// TIA Portal V18 export
FUNCTION "DL_General" : Void   // FC51001, LAD
{ S7_Optimized_Access := 'TRUE' }
VERSION : 0.1
// stored: AutoNumber false, IsIECCheckEnabled false, SetENOAutomatically false, UDAEnableTagReadback false
   VAR_TEMP
      LvlRequest : Array[1..2] of Bool;
      xStopTriger : Bool;
      xCounter1Triger : Bool;
      xCounter2Triger : Bool;
      xPump1ExeriseRun : Bool;
      xPump2ExeriseRun : Bool;
      xPump1ExeriseRunTriger : Bool;
      xPump2ExeriseRunTriger : Bool;
      tTimeExericePump1 : Time;
      tTimeExericePump2 : Time;
   END_VAR
   VAR_TEMP   // added for the SCL form of the ladder/FBD networks
      _w1 : Bool;
      _w2 : Bool;
      _w3 : Bool;
      _w4 : Bool;
      _w5 : Bool;
      _w6 : Bool;
   END_VAR
BEGIN

REGION Network 1 (SCL): PanelModeSelector
   IF "DLsDI".Requests.xDieselLinePumpPanelSelectorAuto THEN
       "DL_Vars".Vars.cDLPanelModeSelector := 3;
   ELSIF "DLsDI".Requests.xDieselLinePumpPanelSelectorP1Man THEN
       "DL_Vars".Vars.cDLPanelModeSelector := 1;
   ELSIF "DLsDI".Requests.xDieselLinePumpPanelSelectorP2Man THEN
       "DL_Vars".Vars.cDLPanelModeSelector := 2;
   ELSIF "DLsDI".Requests.xDieselLinePumpPanelSelectorOff THEN
       "DL_Vars".Vars.cDLPanelModeSelector := 0;
   END_IF;
END_REGION

REGION Network 2
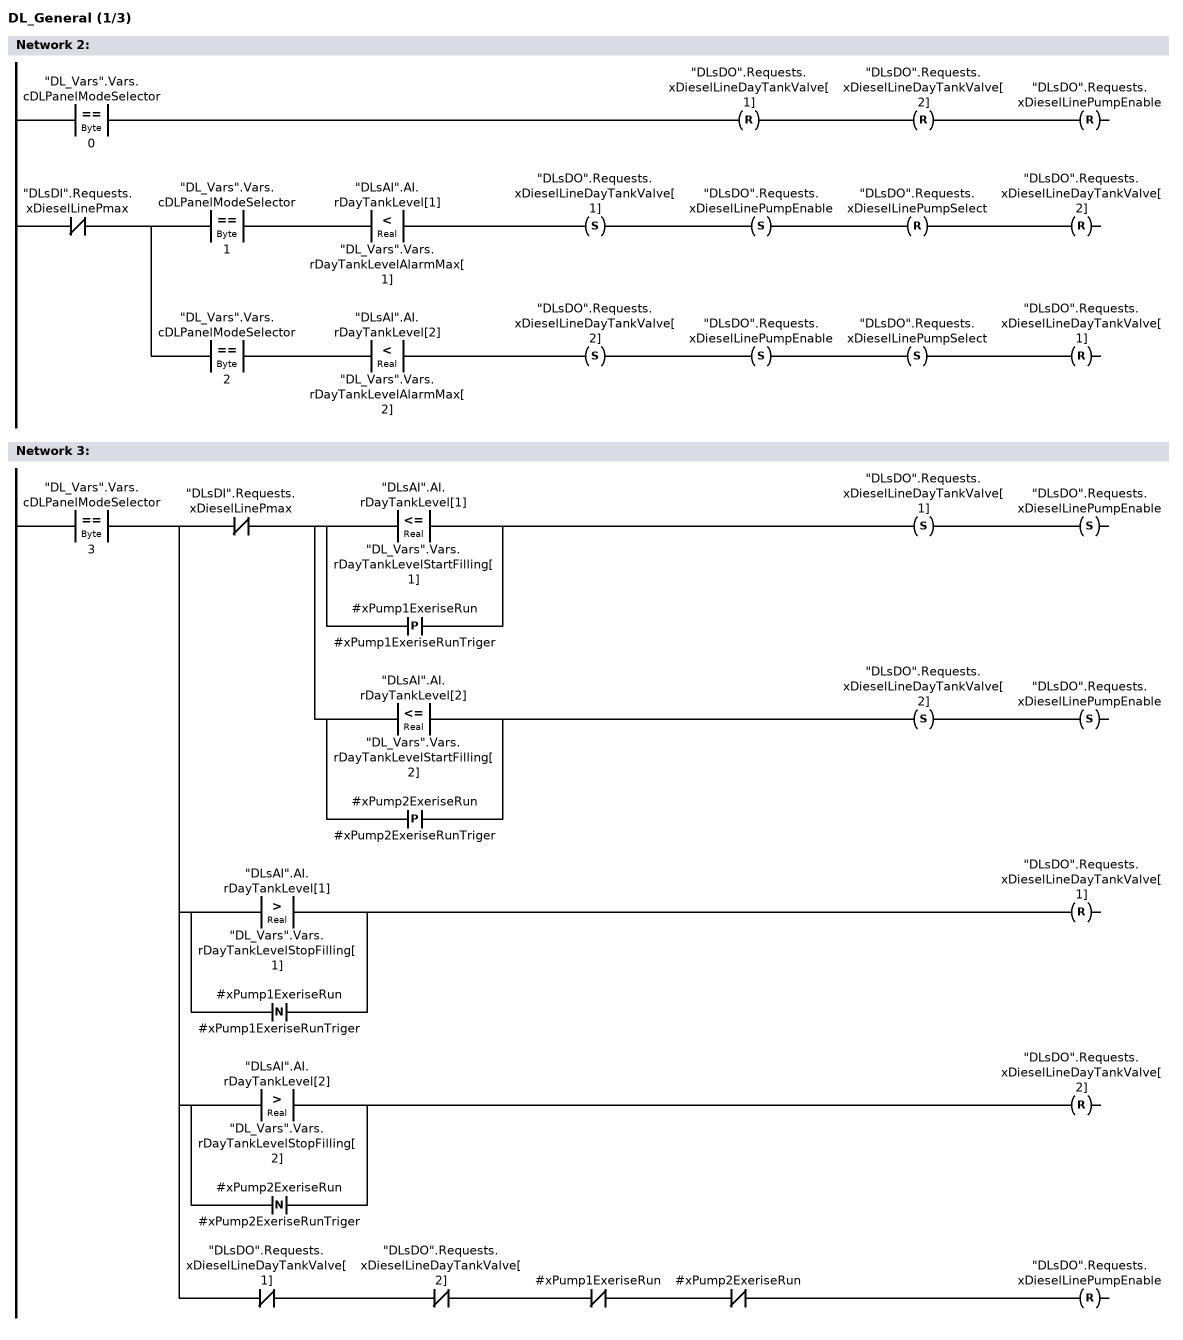
   RUNG wire#powerrail
      { S7_Templates := "SrcType := Byte" } EQ_Contact(in1 := "DL_Vars".Vars.cDLPanelModeSelector, in2 := 0)
      R_Coil( "DLsDO".Requests.xDieselLineDayTankValve[1] )
      R_Coil( "DLsDO".Requests.xDieselLineDayTankValve[2] )
      R_Coil( "DLsDO".Requests.xDieselLinePumpEnable )
   END_RUNG
   RUNG wire#powerrail
      I_Contact( "DLsDI".Requests.xDieselLinePmax )
      wire#w1
      { S7_Templates := "SrcType := Byte" } EQ_Contact(in1 := "DL_Vars".Vars.cDLPanelModeSelector, in2 := 1)
      { S7_Templates := "SrcType := Real" } LT_Contact(in1 := "DLsAI".AI.rDayTankLevel[1], in2 := "DL_Vars".Vars.rDayTankLevelAlarmMax[1])
      S_Coil( "DLsDO".Requests.xDieselLineDayTankValve[1] )
      S_Coil( "DLsDO".Requests.xDieselLinePumpEnable )
      R_Coil( "DLsDO".Requests.xDieselLinePumpSelect )
      R_Coil( "DLsDO".Requests.xDieselLineDayTankValve[2] )
   END_RUNG
   RUNG wire#w1
      { S7_Templates := "SrcType := Byte" } EQ_Contact(in1 := "DL_Vars".Vars.cDLPanelModeSelector, in2 := 2)
      { S7_Templates := "SrcType := Real" } LT_Contact(in1 := "DLsAI".AI.rDayTankLevel[2], in2 := "DL_Vars".Vars.rDayTankLevelAlarmMax[2])
      S_Coil( "DLsDO".Requests.xDieselLineDayTankValve[2] )
      S_Coil( "DLsDO".Requests.xDieselLinePumpEnable )
      S_Coil( "DLsDO".Requests.xDieselLinePumpSelect )
      R_Coil( "DLsDO".Requests.xDieselLineDayTankValve[1] )
   END_RUNG
   // the same network as SCL:
   IF "DL_Vars".Vars.cDLPanelModeSelector = 0 THEN
       "DLsDO".Requests.xDieselLineDayTankValve[1] := FALSE;
       "DLsDO".Requests.xDieselLineDayTankValve[2] := FALSE;
       "DLsDO".Requests.xDieselLinePumpEnable := FALSE;
   END_IF;
   #_w1 := NOT "DLsDI".Requests.xDieselLinePmax;
   IF #_w1 AND ("DL_Vars".Vars.cDLPanelModeSelector = 1) AND ("DLsAI".AI.rDayTankLevel[1] < "DL_Vars".Vars.rDayTankLevelAlarmMax[1]) THEN
       "DLsDO".Requests.xDieselLineDayTankValve[1] := TRUE;
       "DLsDO".Requests.xDieselLinePumpEnable := TRUE;
       "DLsDO".Requests.xDieselLinePumpSelect := FALSE;
       "DLsDO".Requests.xDieselLineDayTankValve[2] := FALSE;
   END_IF;
   IF #_w1 AND ("DL_Vars".Vars.cDLPanelModeSelector = 2) AND ("DLsAI".AI.rDayTankLevel[2] < "DL_Vars".Vars.rDayTankLevelAlarmMax[2]) THEN
       "DLsDO".Requests.xDieselLineDayTankValve[2] := TRUE;
       "DLsDO".Requests.xDieselLinePumpEnable := TRUE;
       "DLsDO".Requests.xDieselLinePumpSelect := TRUE;
       "DLsDO".Requests.xDieselLineDayTankValve[1] := FALSE;
   END_IF;
END_REGION

REGION Network 3
   RUNG wire#powerrail
      { S7_Templates := "SrcType := Byte" } EQ_Contact(in1 := "DL_Vars".Vars.cDLPanelModeSelector, in2 := 3)
      wire#w1
      I_Contact( "DLsDI".Requests.xDieselLinePmax )
      wire#w2
      { S7_Templates := "SrcType := Real" } LE_Contact(in1 := "DLsAI".AI.rDayTankLevel[1], in2 := "DL_Vars".Vars.rDayTankLevelStartFilling[1])
      wire#w3
      S_Coil( "DLsDO".Requests.xDieselLineDayTankValve[1] )
      S_Coil( "DLsDO".Requests.xDieselLinePumpEnable )
   END_RUNG
   RUNG wire#w2
      P_Contact(operand := #xPump1ExeriseRun, bit := #xPump1ExeriseRunTriger)
   END_RUNG wire#w3
   RUNG wire#w2
      { S7_Templates := "SrcType := Real" } LE_Contact(in1 := "DLsAI".AI.rDayTankLevel[2], in2 := "DL_Vars".Vars.rDayTankLevelStartFilling[2])
      wire#w4
      S_Coil( "DLsDO".Requests.xDieselLineDayTankValve[2] )
      S_Coil( "DLsDO".Requests.xDieselLinePumpEnable )
   END_RUNG
   RUNG wire#w2
      P_Contact(operand := #xPump2ExeriseRun, bit := #xPump2ExeriseRunTriger)
   END_RUNG wire#w4
   RUNG wire#w1
      { S7_Templates := "SrcType := Real" } GT_Contact(in1 := "DLsAI".AI.rDayTankLevel[1], in2 := "DL_Vars".Vars.rDayTankLevelStopFilling[1])
      wire#w5
      R_Coil( "DLsDO".Requests.xDieselLineDayTankValve[1] )
   END_RUNG
   RUNG wire#w1
      N_Contact(operand := #xPump1ExeriseRun, bit := #xPump1ExeriseRunTriger)
   END_RUNG wire#w5
   RUNG wire#w1
      { S7_Templates := "SrcType := Real" } GT_Contact(in1 := "DLsAI".AI.rDayTankLevel[2], in2 := "DL_Vars".Vars.rDayTankLevelStopFilling[2])
      wire#w6
      R_Coil( "DLsDO".Requests.xDieselLineDayTankValve[2] )
   END_RUNG
   RUNG wire#w1
      N_Contact(operand := #xPump2ExeriseRun, bit := #xPump2ExeriseRunTriger)
   END_RUNG wire#w6
   RUNG wire#w1
      I_Contact( "DLsDO".Requests.xDieselLineDayTankValve[1] )
      I_Contact( "DLsDO".Requests.xDieselLineDayTankValve[2] )
      I_Contact( #xPump1ExeriseRun )
      I_Contact( #xPump2ExeriseRun )
      R_Coil( "DLsDO".Requests.xDieselLinePumpEnable )
   END_RUNG
   // the same network as SCL:
   #_w1 := "DL_Vars".Vars.cDLPanelModeSelector = 3;
   #_w2 := #_w1 AND NOT "DLsDI".Requests.xDieselLinePmax;
   #_w3 := #_w2 AND #xPump1ExeriseRun AND NOT #xPump1ExeriseRunTriger;   // rising edge of #xPump1ExeriseRun
   #xPump1ExeriseRunTriger := #xPump1ExeriseRun;
   IF (#_w2 AND ("DLsAI".AI.rDayTankLevel[1] <= "DL_Vars".Vars.rDayTankLevelStartFilling[1])) OR #_w3 THEN
       "DLsDO".Requests.xDieselLineDayTankValve[1] := TRUE;
       "DLsDO".Requests.xDieselLinePumpEnable := TRUE;
   END_IF;
   #_w4 := #_w2 AND #xPump2ExeriseRun AND NOT #xPump2ExeriseRunTriger;   // rising edge of #xPump2ExeriseRun
   #xPump2ExeriseRunTriger := #xPump2ExeriseRun;
   IF (#_w2 AND ("DLsAI".AI.rDayTankLevel[2] <= "DL_Vars".Vars.rDayTankLevelStartFilling[2])) OR #_w4 THEN
       "DLsDO".Requests.xDieselLineDayTankValve[2] := TRUE;
       "DLsDO".Requests.xDieselLinePumpEnable := TRUE;
   END_IF;
   #_w5 := #_w1 AND NOT #xPump1ExeriseRun AND #xPump1ExeriseRunTriger;   // falling edge of #xPump1ExeriseRun
   #xPump1ExeriseRunTriger := #xPump1ExeriseRun;
   IF (#_w1 AND ("DLsAI".AI.rDayTankLevel[1] > "DL_Vars".Vars.rDayTankLevelStopFilling[1])) OR #_w5 THEN
       "DLsDO".Requests.xDieselLineDayTankValve[1] := FALSE;
   END_IF;
   #_w6 := #_w1 AND NOT #xPump2ExeriseRun AND #xPump2ExeriseRunTriger;   // falling edge of #xPump2ExeriseRun
   #xPump2ExeriseRunTriger := #xPump2ExeriseRun;
   IF (#_w1 AND ("DLsAI".AI.rDayTankLevel[2] > "DL_Vars".Vars.rDayTankLevelStopFilling[2])) OR #_w6 THEN
       "DLsDO".Requests.xDieselLineDayTankValve[2] := FALSE;
   END_IF;
   IF #_w1 AND NOT "DLsDO".Requests.xDieselLineDayTankValve[1] AND NOT "DLsDO".Requests.xDieselLineDayTankValve[2] AND NOT #xPump1ExeriseRun AND NOT #xPump2ExeriseRun THEN
       "DLsDO".Requests.xDieselLinePumpEnable := FALSE;
   END_IF;
END_REGION

REGION Network 4
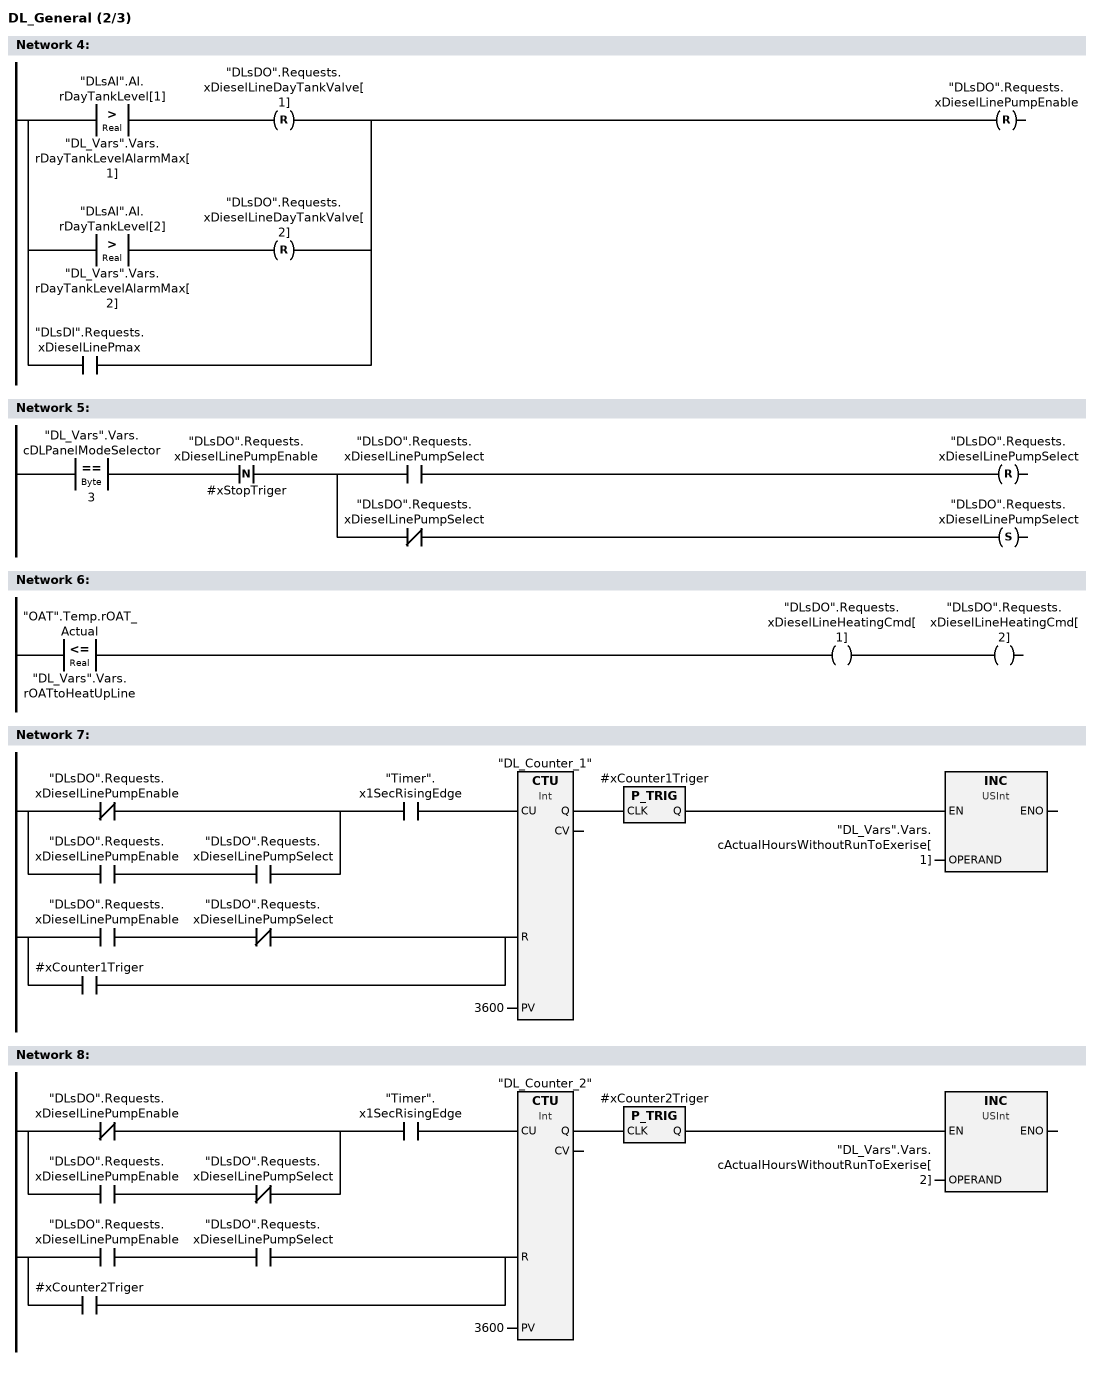
   RUNG wire#powerrail
      { S7_Templates := "SrcType := Real" } GT_Contact(in1 := "DLsAI".AI.rDayTankLevel[1], in2 := "DL_Vars".Vars.rDayTankLevelAlarmMax[1])
      R_Coil( "DLsDO".Requests.xDieselLineDayTankValve[1] )
      wire#w1
      R_Coil( "DLsDO".Requests.xDieselLinePumpEnable )
   END_RUNG
   RUNG wire#powerrail
      { S7_Templates := "SrcType := Real" } GT_Contact(in1 := "DLsAI".AI.rDayTankLevel[2], in2 := "DL_Vars".Vars.rDayTankLevelAlarmMax[2])
      R_Coil( "DLsDO".Requests.xDieselLineDayTankValve[2] )
   END_RUNG wire#w1
   RUNG wire#powerrail
      Contact( "DLsDI".Requests.xDieselLinePmax )
   END_RUNG wire#w1
   // the same network as SCL:
   #_w1 := "DLsAI".AI.rDayTankLevel[1] > "DL_Vars".Vars.rDayTankLevelAlarmMax[1];
   IF #_w1 THEN "DLsDO".Requests.xDieselLineDayTankValve[1] := FALSE; END_IF;
   #_w2 := "DLsAI".AI.rDayTankLevel[2] > "DL_Vars".Vars.rDayTankLevelAlarmMax[2];
   IF #_w2 THEN "DLsDO".Requests.xDieselLineDayTankValve[2] := FALSE; END_IF;
   IF #_w1 OR #_w2 OR "DLsDI".Requests.xDieselLinePmax THEN
       "DLsDO".Requests.xDieselLinePumpEnable := FALSE;
   END_IF;
END_REGION

REGION Network 5
   RUNG wire#powerrail
      { S7_Templates := "SrcType := Byte" } EQ_Contact(in1 := "DL_Vars".Vars.cDLPanelModeSelector, in2 := 3)
      N_Contact(operand := "DLsDO".Requests.xDieselLinePumpEnable, bit := #xStopTriger)
      wire#w1
      Contact( "DLsDO".Requests.xDieselLinePumpSelect )
      R_Coil( "DLsDO".Requests.xDieselLinePumpSelect )
   END_RUNG
   RUNG wire#w1
      I_Contact( "DLsDO".Requests.xDieselLinePumpSelect )
      S_Coil( "DLsDO".Requests.xDieselLinePumpSelect )
   END_RUNG
   // the same network as SCL:
   #_w1 := ("DL_Vars".Vars.cDLPanelModeSelector = 3) AND NOT "DLsDO".Requests.xDieselLinePumpEnable AND #xStopTriger;   // falling edge of "DLsDO".Requests.xDieselLinePumpEnable
   #xStopTriger := "DLsDO".Requests.xDieselLinePumpEnable;
   IF #_w1 AND "DLsDO".Requests.xDieselLinePumpSelect THEN
       "DLsDO".Requests.xDieselLinePumpSelect := FALSE;
   END_IF;
   IF #_w1 AND NOT "DLsDO".Requests.xDieselLinePumpSelect THEN
       "DLsDO".Requests.xDieselLinePumpSelect := TRUE;
   END_IF;
END_REGION

REGION Network 6
   RUNG wire#powerrail
      { S7_Templates := "SrcType := Real" } LE_Contact(in1 := "OAT".Temp.rOAT_Actual, in2 := "DL_Vars".Vars.rOATtoHeatUpLine)
      Coil( "DLsDO".Requests.xDieselLineHeatingCmd[1] )
      Coil( "DLsDO".Requests.xDieselLineHeatingCmd[2] )
   END_RUNG
   // the same network as SCL:
   "DLsDO".Requests.xDieselLineHeatingCmd[1] := "OAT".Temp.rOAT_Actual <= "DL_Vars".Vars.rOATtoHeatUpLine;
   "DLsDO".Requests.xDieselLineHeatingCmd[2] := "OAT".Temp.rOAT_Actual <= "DL_Vars".Vars.rOATtoHeatUpLine;
END_REGION

REGION Network 7
   RUNG wire#powerrail
      I_Contact( "DLsDO".Requests.xDieselLinePumpEnable )
      wire#w1
      Contact( "Timer".x1SecRisingEdge )
      { S7_Templates := "value_type := Int" } "DL_Counter_1".CTU(r := wire#w2, pv := 3600, cv =>)
      P_Trig( #xCounter1Triger )
      { S7_Templates := "DestType := USInt" } Inc( "DL_Vars".Vars.cActualHoursWithoutRunToExerise[1] )
   END_RUNG
   RUNG wire#powerrail
      Contact( "DLsDO".Requests.xDieselLinePumpEnable )
      Contact( "DLsDO".Requests.xDieselLinePumpSelect )
   END_RUNG wire#w1
   RUNG wire#powerrail
      Contact( "DLsDO".Requests.xDieselLinePumpEnable )
      I_Contact( "DLsDO".Requests.xDieselLinePumpSelect )
   END_RUNG wire#w2
   RUNG wire#powerrail
      Contact( #xCounter1Triger )
   END_RUNG wire#w2
   // the same network as SCL:
   "DL_Counter_1".CTU(CU := (NOT "DLsDO".Requests.xDieselLinePumpEnable OR ("DLsDO".Requests.xDieselLinePumpEnable AND "DLsDO".Requests.xDieselLinePumpSelect)) AND "Timer".x1SecRisingEdge,
                      R := ("DLsDO".Requests.xDieselLinePumpEnable AND NOT "DLsDO".Requests.xDieselLinePumpSelect) OR #xCounter1Triger,
                      PV := 3600);
   #_w1 := "DL_Counter_1".Q AND NOT #xCounter1Triger;   // rising edge
   #xCounter1Triger := "DL_Counter_1".Q;
   IF #_w1 THEN
       "DL_Vars".Vars.cActualHoursWithoutRunToExerise[1] := "DL_Vars".Vars.cActualHoursWithoutRunToExerise[1] + 1;
   END_IF;
END_REGION

REGION Network 8
   RUNG wire#powerrail
      I_Contact( "DLsDO".Requests.xDieselLinePumpEnable )
      wire#w1
      Contact( "Timer".x1SecRisingEdge )
      { S7_Templates := "value_type := Int" } "DL_Counter_2".CTU(r := wire#w2, pv := 3600, cv =>)
      P_Trig( #xCounter2Triger )
      { S7_Templates := "DestType := USInt" } Inc( "DL_Vars".Vars.cActualHoursWithoutRunToExerise[2] )
   END_RUNG
   RUNG wire#powerrail
      Contact( "DLsDO".Requests.xDieselLinePumpEnable )
      I_Contact( "DLsDO".Requests.xDieselLinePumpSelect )
   END_RUNG wire#w1
   RUNG wire#powerrail
      Contact( "DLsDO".Requests.xDieselLinePumpEnable )
      Contact( "DLsDO".Requests.xDieselLinePumpSelect )
   END_RUNG wire#w2
   RUNG wire#powerrail
      Contact( #xCounter2Triger )
   END_RUNG wire#w2
   // the same network as SCL:
   "DL_Counter_2".CTU(CU := (NOT "DLsDO".Requests.xDieselLinePumpEnable OR ("DLsDO".Requests.xDieselLinePumpEnable AND NOT "DLsDO".Requests.xDieselLinePumpSelect)) AND "Timer".x1SecRisingEdge,
                      R := ("DLsDO".Requests.xDieselLinePumpEnable AND "DLsDO".Requests.xDieselLinePumpSelect) OR #xCounter2Triger,
                      PV := 3600);
   #_w1 := "DL_Counter_2".Q AND NOT #xCounter2Triger;   // rising edge
   #xCounter2Triger := "DL_Counter_2".Q;
   IF #_w1 THEN
       "DL_Vars".Vars.cActualHoursWithoutRunToExerise[2] := "DL_Vars".Vars.cActualHoursWithoutRunToExerise[2] + 1;
   END_IF;
END_REGION

REGION Network 9
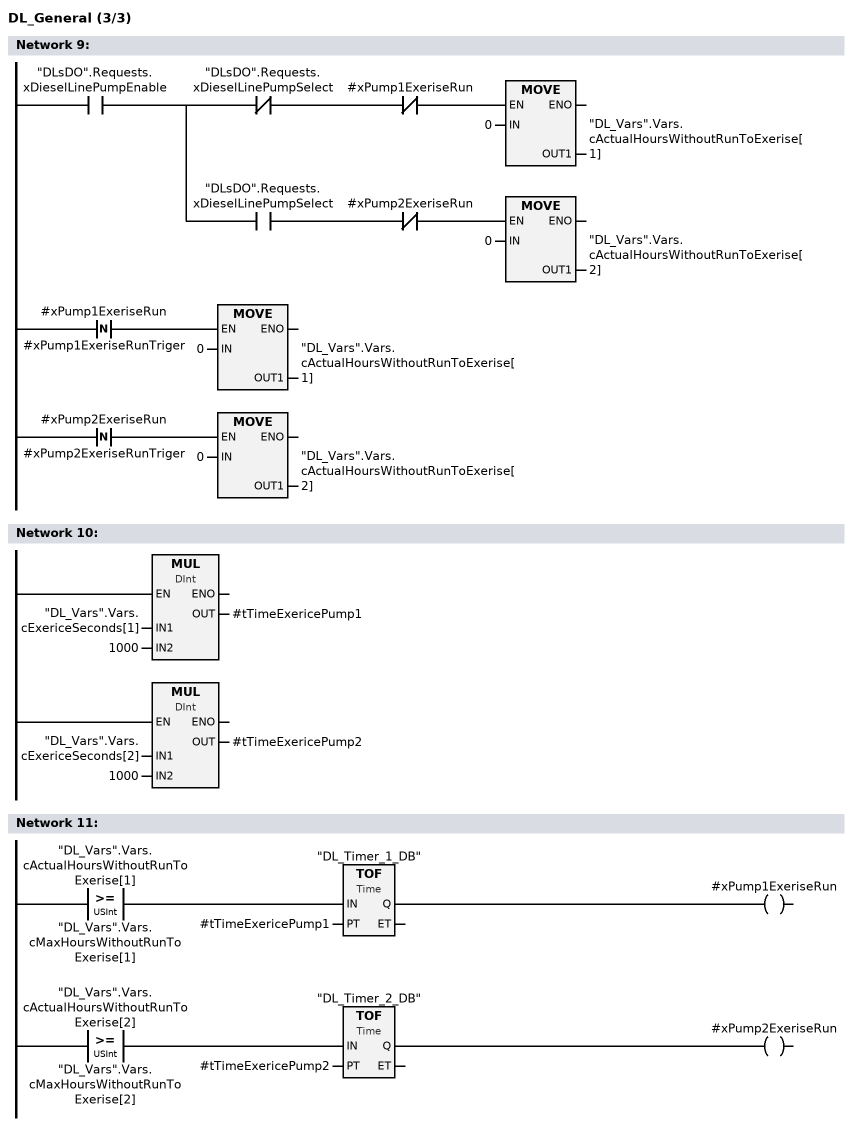
   RUNG wire#powerrail
      Contact( "DLsDO".Requests.xDieselLinePumpEnable )
      wire#w1
      I_Contact( "DLsDO".Requests.xDieselLinePumpSelect )
      I_Contact( #xPump1ExeriseRun )
      Move(in := 0, out1 => "DL_Vars".Vars.cActualHoursWithoutRunToExerise[1])
   END_RUNG
   RUNG wire#w1
      Contact( "DLsDO".Requests.xDieselLinePumpSelect )
      I_Contact( #xPump2ExeriseRun )
      Move(in := 0, out1 => "DL_Vars".Vars.cActualHoursWithoutRunToExerise[2])
   END_RUNG
   RUNG wire#powerrail
      N_Contact(operand := #xPump1ExeriseRun, bit := #xPump1ExeriseRunTriger)
      Move(in := 0, out1 => "DL_Vars".Vars.cActualHoursWithoutRunToExerise[1])
   END_RUNG
   RUNG wire#powerrail
      N_Contact(operand := #xPump2ExeriseRun, bit := #xPump2ExeriseRunTriger)
      Move(in := 0, out1 => "DL_Vars".Vars.cActualHoursWithoutRunToExerise[2])
   END_RUNG
   // the same network as SCL:
   IF "DLsDO".Requests.xDieselLinePumpEnable AND NOT "DLsDO".Requests.xDieselLinePumpSelect AND NOT #xPump1ExeriseRun THEN
       "DL_Vars".Vars.cActualHoursWithoutRunToExerise[1] := 0;
   END_IF;
   IF "DLsDO".Requests.xDieselLinePumpEnable AND "DLsDO".Requests.xDieselLinePumpSelect AND NOT #xPump2ExeriseRun THEN
       "DL_Vars".Vars.cActualHoursWithoutRunToExerise[2] := 0;
   END_IF;
   #_w1 := NOT #xPump1ExeriseRun AND #xPump1ExeriseRunTriger;   // falling edge of #xPump1ExeriseRun
   #xPump1ExeriseRunTriger := #xPump1ExeriseRun;
   IF #_w1 THEN "DL_Vars".Vars.cActualHoursWithoutRunToExerise[1] := 0; END_IF;
   #_w2 := NOT #xPump2ExeriseRun AND #xPump2ExeriseRunTriger;   // falling edge of #xPump2ExeriseRun
   #xPump2ExeriseRunTriger := #xPump2ExeriseRun;
   IF #_w2 THEN "DL_Vars".Vars.cActualHoursWithoutRunToExerise[2] := 0; END_IF;
END_REGION

REGION Network 10
   RUNG wire#powerrail
      { S7_Templates := "SrcType := DInt" } Mul(in1 := "DL_Vars".Vars.cExericeSeconds[1], in2 := 1000, out => #tTimeExericePump1)
   END_RUNG
   RUNG wire#powerrail
      { S7_Templates := "SrcType := DInt" } Mul(in1 := "DL_Vars".Vars.cExericeSeconds[2], in2 := 1000, out => #tTimeExericePump2)
   END_RUNG
   // the same network as SCL:
   #tTimeExericePump1 := "DL_Vars".Vars.cExericeSeconds[1] * 1000;
   #tTimeExericePump2 := "DL_Vars".Vars.cExericeSeconds[2] * 1000;
END_REGION

REGION Network 11
   RUNG wire#powerrail
      { S7_Templates := "SrcType := USInt" } GE_Contact(in1 := "DL_Vars".Vars.cActualHoursWithoutRunToExerise[1], in2 := "DL_Vars".Vars.cMaxHoursWithoutRunToExerise[1])
      { S7_Templates := "time_type := Time" } "DL_Timer_1_DB".TOF(pt := #tTimeExericePump1, et =>)
      Coil( #xPump1ExeriseRun )
   END_RUNG
   RUNG wire#powerrail
      { S7_Templates := "SrcType := USInt" } GE_Contact(in1 := "DL_Vars".Vars.cActualHoursWithoutRunToExerise[2], in2 := "DL_Vars".Vars.cMaxHoursWithoutRunToExerise[2])
      { S7_Templates := "time_type := Time" } "DL_Timer_2_DB".TOF(pt := #tTimeExericePump2, et =>)
      Coil( #xPump2ExeriseRun )
   END_RUNG
   // the same network as SCL:
   "DL_Timer_1_DB".TOF(IN := "DL_Vars".Vars.cActualHoursWithoutRunToExerise[1] >= "DL_Vars".Vars.cMaxHoursWithoutRunToExerise[1],
                       PT := #tTimeExericePump1);
   #xPump1ExeriseRun := "DL_Timer_1_DB".Q;
   "DL_Timer_2_DB".TOF(IN := "DL_Vars".Vars.cActualHoursWithoutRunToExerise[2] >= "DL_Vars".Vars.cMaxHoursWithoutRunToExerise[2],
                       PT := #tTimeExericePump2);
   #xPump2ExeriseRun := "DL_Timer_2_DB".Q;
END_REGION
END_FUNCTION
